{attribute 'linkalways'} 
{attribute 'no_explicit_call' := 'This FB is a CLASS and must be accessed using methods or properties'}
{attribute 'enable_dynamic_creation'}
FUNCTION_BLOCK Node_F_VN_ReverseContainer EXTENDS VisionNode
VAR
    ipContainer : _ITcVnContainer;
    hrPrev : _HRESULT(S_OK);
	hresult : _HRESULT(S_OK);
END_VAR

METHOD PUBLIC  Clone : I_Node
VAR
	pNode : POINTER TO Node_F_VN_ReverseContainer;
END_VAR
pNode := __NEW(Node_F_VN_ReverseContainer);
Clone := pNode^;
END_METHOD

METHOD FB_init : BOOL
VAR_INPUT
	bInitRetains : BOOL; // if TRUE, the retain variables are initialized (warm start / cold start)
	bInCopyCode : BOOL;  // if TRUE, the instance afterwards gets moved into the copy code (online change)
END_VAR
AddInput('ipContainer', ipContainer);
AddInput('hrPrev', hrPrev);
AddOutput('hresult',hresult);
END_METHOD

METHOD PROTECTED OnExecute
hresult.Value := F_VN_ReverseContainer(
	ipContainer := ipContainer.Value,
	hrPrev:= hrPrev.Value);
END_METHOD

METHOD PUBLIC PreExecutionCheck
VAR_INPUT
	Check : I_PreExecutionChecks;
END_VAR
Check.IsTrue(ipContainer.IsValid, 'ipContainer must be a valid container');
END_METHOD

END_FUNCTION_BLOCK

(* stored: Version 1.1.0.1, ProductVersion 3.1.4024.13
   POU Node_F_VN_ReverseContainer: Id {ca9e5c8d-14d0-0904-36e0-f00e1a1c9b5b}, SpecialFunc None
   Folder Constructor: Id {5bcf6d11-a4ce-0d59-089d-66eb04b4e4ba}
   Method Clone: Id {0457956e-1128-059c-001c-75096c0aeb9c}
   Method FB_init: Id {1f01e3b0-253e-048c-3bdd-44c44fac4821}
   Method OnExecute: Id {f3cb073a-4b3f-07fa-025e-f996952fb7f3}
   Method PreExecutionCheck: Id {9d1cc820-23ea-0db1-2919-1f22ddc7e924} *)
